// TIA Portal V17 export
// export: Created 2024-08-20T10:59:38.4257415Z, ExportSetting WithDefaults, DisplayName Totally Integrated Automation Portal, DisplayVersion V17 Update 4, DisplayName TIA Portal Openness, DisplayVersion V17 Update 4, DisplayName TIA Portal Version Control Interface, DisplayVersion V17, DisplayName STEP 7 Professional, DisplayVersion V17 Update 4, DisplayName STEP 7 Safety, DisplayVersion V17, DisplayName WinCC Advanced, DisplayVersion V17 Update 4
FUNCTION_BLOCK "INSTRUMENTO"   // FB201, LAD
TITLE = BLOCO PARA CONVERSÃO DE ESCALA DE ENGENHARIA
{ S7_Optimized_Access := 'FALSE' }
VERSION : 0.1
// stored: AutoNumber false, IsIECCheckEnabled false, SetENOAutomatically false, UDAEnableTagReadback false
   VAR_INPUT
      "VALOR MANUAL" : Real;   // VALOR MANUAL (HMI)
      EA : Int;   // LEITURA DO CANAL ANALÓGICO
      EA_IE : Real;   // INÍCIO DA ESCALA DO CANAL
      EA_FE : Real;   // FIM DE ESCALA DO CANAL
      S_IE : Real;   // INÍCIO DE ESCALA DE ENGENHARIA PRINCIPAL
      S_FE : Real;   // FIM DE ESCALA DE ENGENHARIA PRINCIPAL
      S2_IE : Real;   // INÍCIO DE ESCALA DE ENGENHARIA SECUNDÁRIA
      S2_FE : Real;   // FIM DE ESCALA DE ENGENHARIA SECUNDÁRIA
      SPLL : Real;   // SETPOINT MUITO BAIXO
      SPL : Real;   // SETPOINT BAIXO
      SPH : Real;   // SETPOINT ALTO
      SPHH : Real;   // SETPOINT MUITO ALTO
      TE_LL : Time;   // DELAY PARA ALARME MUITO BAIXO
      TE_L : Time;   // DELAY PARA ALARME BAIXO
      TE_H : Time;   // DELAY PARA ALARME ALTO
      TE_HH : Time;   // DELAY PARA ALARME MUITO ALTO
      FRH : Int;   // VALOR ALTO PARA ALARME DE FALHA DE LEITURA
      FRL : Int;   // VALOR BAIXO PARA ALARME DE FALHA DE LEITURA
      LIM : Bool;   // LIMITA O VALOR À ESCALA
      MANUAL : Bool;   // HABILITA MANUTENÇÃO DO INSTRUMENTO
      COND : Bool;   // CONDIÇÃO PARA GERAR ALARME
      SPR_YLL : Bool;   // HABILITA SUPRESSÃO ALARME MUITO BAIXO
      SPR_YL : Bool;   // HABILITA SUPRESSÃO ALARME BAIXO
      SPR_YH : Bool;   // HABILITA SUPRESSÃO ALARME ALTO
      SPR_YHH : Bool;   // HABILITA SUPRESSÃO ALARME MUITO ALTO
   END_VAR
   VAR_OUTPUT
      VNP : Real;   // VALOR CONVERTIDO PARA ESCALA DE ENGENHARIA PRINCIPAL
      YLL : Bool;   // ALARME MUITO BAIXO
      YL : Bool;   // ALARME BAIXO
      YH : Bool;   // ALARME ALTO
      YHH : Bool;   // ALARME MUITO ALTO
      YF : Bool;   // ALARME DE FALHA NA MEDIÇÃO
      VNS : Real;   // VALOR CONVERTIDO PARA ESCALA DE ENGENHARIA SECUNDÁRIA
      LL : Bool;   // VALOR MUITO BAIXO
      L : Bool;   // VALOR BAIXO
      H : Bool;   // VALOR ALTO
      HH : Bool;   // VALOR MUITO ALTO
   END_VAR
   VAR DB_SPECIFIC
      TLL { S7_SetPoint := 'True'} : TON_TIME;   // TEMPO PARA GERAR ALARME
      TL { S7_SetPoint := 'True'} : TON_TIME;   // TEMPO PARA GERAR ALARME
      TH { S7_SetPoint := 'True'} : TON_TIME;   // TEMPO PARA GERAR ALARME
      THH { S7_SetPoint := 'True'} : TON_TIME;   // TEMPO PARA GERAR ALARME
      FALHA : Bool;   // SINALIZAÇÃO DE FALHA NO INSTRUMENTO
   END_VAR
   VAR_TEMP
      EAR : Real;   // VALOR LIDO DA ENTRADA ANALÓGICA
      AC01 : Real;   // AUXILIAR PARA CÁLCULO
      AC02 : Real;   // AUXILIAR PARA CÁLCULO
      AC03 : Real;   // AUXILIAR PARA CÁLCULO
      AC04 : Real;   // AUXILIAR PARA CÁLCULO
      AC05 : Real;   // AUXILIAR PARA CÁLCULO
      AC06 : Real;   // AUXILIAR PARA CÁLCULO
      AC07 : Real;   // AUXILIAR PARA CÁLCULO
      AC08 : Real;   // AUXILIAR PARA CÁLCULO
      AC09 : Real;   // AUXILIAR PARA CÁLCULO
      AC10 : Real;   // AUXILIAR PARA CÁLCULO
      RESULT_P : Real;   // RESULTADO DA ESCALA
      RESULT_S : Real;   // RESULTADO DA ESCALA
      ET_TLL : Time;   // EFETIVO DO TEMPORIZADOR
      ET_TL : Time;   // EFETIVO DO TEMPORIZADOR
      ET_TH : Time;   // EFETIVO DO TEMPORIZADOR
      ET_THH : Time;   // EFETIVO DO TEMPORIZADOR
      EADI : DInt;
   END_VAR
BEGIN

REGION Network 1: CONVERSOR O VALOR LIDO DO CARTÃO PARA REAL
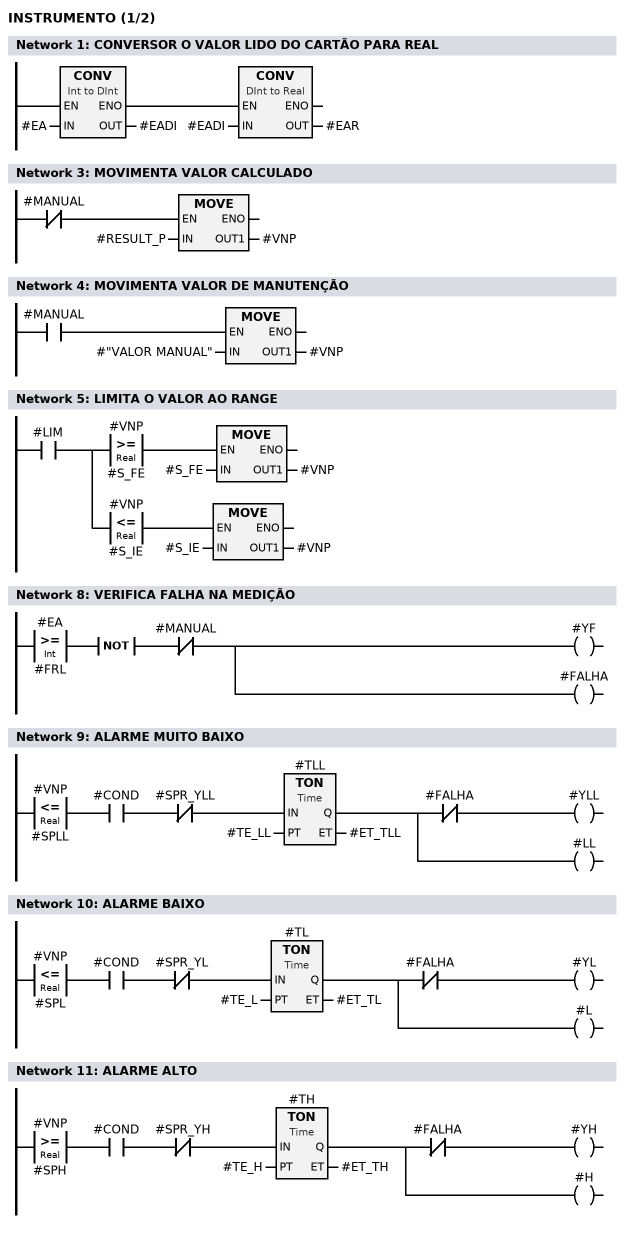
   RUNG wire#powerrail
      { S7_Templates := "[SrcType := Int, DestType := DInt]"; S7_GenerateENO := "TRUE" } Convert(in := #EA, out => #EADI)
      { S7_Templates := "[SrcType := DInt, DestType := Real]"; S7_GenerateENO := "TRUE" } Convert(in := #EADI, out => #EAR)
   END_RUNG
   // the same network as SCL:
   // ENO of a box is taken as its EN; it also drops when the box reports an error
   #EADI := INT_TO_DINT(#EA);
   #EAR := DINT_TO_REAL(#EADI);
END_REGION

NETWORK
TITLE = CONVERTER PARA ESCALA DE ENGENHARIA PRINCIPAL
      L     #EAR;
      L     #EA_IE;
      -R;
      T     #AC01;

      L     #S_FE;  // Subtrai escalas de saída
      L     #S_IE;
      -R;
      T     #AC02;

      L     #EA_FE;  // Subtrai escalas de entrada
      L     #EA_IE;
      -R;
      T     #AC03;

      L     #AC01;  // Multiplica resultado das subtrações
      L     #AC02;
      *R;
      T     #AC04;

      L     #AC04;  // Divide o produto pela subtração das escalas de entrada
      L     #AC03;
      /R;
      T     #AC05;

      L     #AC05;  // Soma o valor de fim da escala de saída
      L     #S_IE;
      +R;
      T     #RESULT_P;  // Resultado do cálculo
      T     #VNP;  // Transfere valor já convertido


REGION Network 3: MOVIMENTA VALOR CALCULADO
   RUNG wire#powerrail
      I_Contact( #MANUAL )
      Move(in := #RESULT_P, out1 => #VNP)
   END_RUNG
   // the same network as SCL:
   IF NOT #MANUAL THEN #VNP := #RESULT_P; END_IF;
END_REGION

REGION Network 4: MOVIMENTA VALOR DE MANUTENÇÃO
   RUNG wire#powerrail
      Contact( #MANUAL )
      Move(in := #"VALOR MANUAL", out1 => #VNP)
   END_RUNG
   // the same network as SCL:
   IF #MANUAL THEN #VNP := #"VALOR MANUAL"; END_IF;
END_REGION

REGION Network 5: LIMITA O VALOR AO RANGE
   RUNG wire#powerrail
      Contact( #LIM )
      wire#w1
      { S7_Templates := "SrcType := Real" } GE_Contact(in1 := #VNP, in2 := #S_FE)
      { S7_GenerateENO := "TRUE" } Move(in := #S_FE, out1 => #VNP)
   END_RUNG
   RUNG wire#w1
      { S7_Templates := "SrcType := Real" } LE_Contact(in1 := #VNP, in2 := #S_IE)
      { S7_GenerateENO := "TRUE" } Move(in := #S_IE, out1 => #VNP)
   END_RUNG
   // the same network as SCL:
   IF #LIM AND (#VNP >= #S_FE) THEN #VNP := #S_FE; END_IF;
   IF #LIM AND (#VNP <= #S_IE) THEN #VNP := #S_IE; END_IF;
END_REGION

NETWORK
TITLE = MOVIMENTA 0 PARA A LEITURA
      A     #YF;
      AN    #MANUAL;
      JNB   _004;
      L     0;
      T     #VNP;
_004: NOP   0;

NETWORK
TITLE = CONVERTER PARA ESCALA DE ENGENHARIA SECUNDÁRIA
      L     #VNP;
      L     #S_IE;
      -R;
      T     #AC06;

      L     #S2_FE;  // Subtrai escalas de saída
      L     #S2_IE;
      -R;
      T     #AC07;

      L     #S_FE;  // Subtrai escalas de entrada
      L     #S_IE;
      -R;
      T     #AC08;

      L     #AC06;  // Multiplica resultado das subtrações
      L     #AC07;
      *R;
      T     #AC09;

      L     #AC09;  // Divide o produto pela subtração das escalas de entrada
      L     #AC08;
      /R;
      T     #AC10;

      L     #AC10;  // Soma o valor de fim da escala de saída
      L     #S2_IE;
      +R;
      T     #RESULT_S;  // Resultado do cálculo
      T     #VNS;  // Transfere valor já convertido


REGION Network 8: VERIFICA FALHA NA MEDIÇÃO
   RUNG wire#powerrail
      { S7_Templates := "SrcType := Int" } GE_Contact(in1 := #EA, in2 := #FRL)
      Not()
      I_Contact( #MANUAL )
      wire#w1
      Coil( #YF )
   END_RUNG
   RUNG wire#w1
      Coil( #FALHA )
   END_RUNG
   // the same network as SCL:
   #YF := NOT (#EA >= #FRL) AND NOT #MANUAL;
   #FALHA := #YF;
END_REGION

REGION Network 9: ALARME MUITO BAIXO
   RUNG wire#powerrail
      { S7_Templates := "SrcType := Real" } LE_Contact(in1 := #VNP, in2 := #SPLL)
      Contact( #COND )
      I_Contact( #SPR_YLL )
      { S7_Templates := "time_type := Time" } #TLL.TON(pt := #TE_LL, et => #ET_TLL)
      wire#w1
      I_Contact( #FALHA )
      Coil( #YLL )
   END_RUNG
   RUNG wire#w1
      Coil( #LL )
   END_RUNG
   // the same network as SCL:
   #TLL(IN := (#VNP <= #SPLL) AND #COND AND NOT #SPR_YLL, PT := #TE_LL, ET => #ET_TLL);   // TON
   #YLL := #TLL.Q AND NOT #FALHA;
   #LL := #TLL.Q;
END_REGION

REGION Network 10: ALARME BAIXO
   RUNG wire#powerrail
      { S7_Templates := "SrcType := Real" } LE_Contact(in1 := #VNP, in2 := #SPL)
      Contact( #COND )
      I_Contact( #SPR_YL )
      { S7_Templates := "time_type := Time" } #TL.TON(pt := #TE_L, et => #ET_TL)
      wire#w1
      I_Contact( #FALHA )
      Coil( #YL )
   END_RUNG
   RUNG wire#w1
      Coil( #L )
   END_RUNG
   // the same network as SCL:
   #TL(IN := (#VNP <= #SPL) AND #COND AND NOT #SPR_YL, PT := #TE_L, ET => #ET_TL);   // TON
   #YL := #TL.Q AND NOT #FALHA;
   #L := #TL.Q;
END_REGION

REGION Network 11: ALARME ALTO
   RUNG wire#powerrail
      { S7_Templates := "SrcType := Real" } GE_Contact(in1 := #VNP, in2 := #SPH)
      Contact( #COND )
      I_Contact( #SPR_YH )
      { S7_Templates := "time_type := Time" } #TH.TON(pt := #TE_H, et => #ET_TH)
      wire#w1
      I_Contact( #FALHA )
      Coil( #YH )
   END_RUNG
   RUNG wire#w1
      Coil( #H )
   END_RUNG
   // the same network as SCL:
   #TH(IN := (#VNP >= #SPH) AND #COND AND NOT #SPR_YH, PT := #TE_H, ET => #ET_TH);   // TON
   #YH := #TH.Q AND NOT #FALHA;
   #H := #TH.Q;
END_REGION

REGION Network 12: ALARME MUITO ALTO
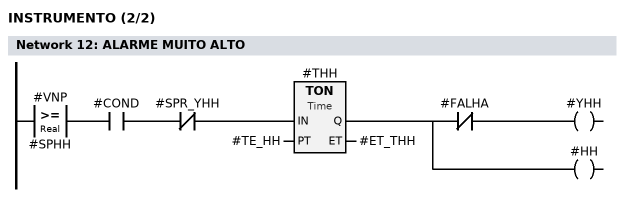
   RUNG wire#powerrail
      { S7_Templates := "SrcType := Real" } GE_Contact(in1 := #VNP, in2 := #SPHH)
      Contact( #COND )
      I_Contact( #SPR_YHH )
      { S7_Templates := "time_type := Time" } #THH.TON(pt := #TE_HH, et => #ET_THH)
      wire#w1
      I_Contact( #FALHA )
      Coil( #YHH )
   END_RUNG
   RUNG wire#w1
      Coil( #HH )
   END_RUNG
   // the same network as SCL:
   #THH(IN := (#VNP >= #SPHH) AND #COND AND NOT #SPR_YHH, PT := #TE_HH, ET => #ET_THH);   // TON
   #YHH := #THH.Q AND NOT #FALHA;
   #HH := #THH.Q;
END_REGION
END_FUNCTION_BLOCK
